TYPE ST_FeedbackOneType :
STRUCT
	Manufacturer : E_Manufacturer;



END_STRUCT
END_TYPE

(* stored: Version 1.1.0.1, ProductVersion 3.1.4024.12
   DUT ST_FeedbackOneType: Id {9dd148a8-7d6a-4bbc-98f0-6a1986e0fcb4} *)
